TYPE ST_PlcInfo :
STRUCT
	sTargetType 	: STRING(30);
	sSerialNo 		: STRING(16);
	sTwinCATBuild 	: STRING(8);
	sPlcVersion		: STRING(10);
END_STRUCT
END_TYPE

(* stored: Version 1.1.0.1, ProductVersion 3.1.4022.12
   DUT ST_PlcInfo: Id {453e4874-e616-41ee-8f2a-f2f5369dc0e5} *)
